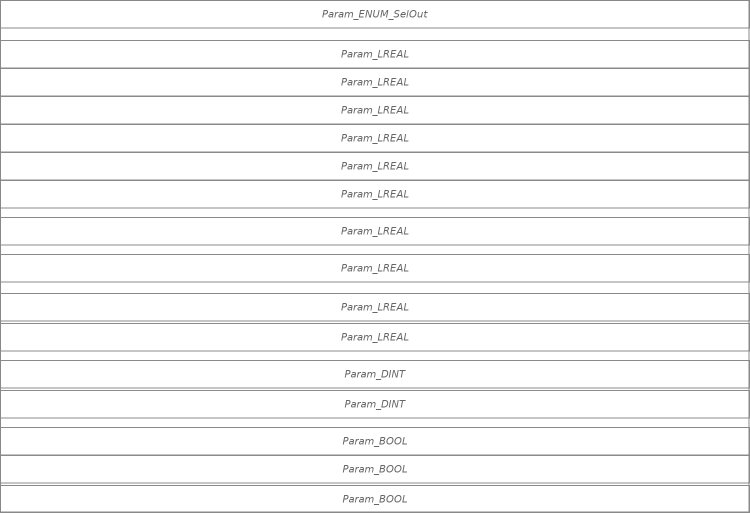
VISUALIZATION Visu_Mparam_Cool  // 750x513
    Frame (0,40 750x28)
        shows Param_LREAL(nIdx := 4)
    Frame (0,68 750x28)
        shows Param_LREAL(nIdx := 6)
    Frame (0,96 750x28)
        shows Param_LREAL(nIdx := 8)
    Frame (0,124 750x28)
        shows Param_LREAL(nIdx := 10)
    Frame (0,360 750x28)
        shows Param_DINT(nIdx := 11)
    Frame (0,0 750x28)
        shows Param_ENUM_SelOut(nIdx := GlobalOne)
    Frame (0,152 750x28)
        shows Param_LREAL(nIdx := 16)
    Frame (0,180 750x28)
        shows Param_LREAL(nIdx := 17)
    Frame (0,217 750x28)
        shows Param_LREAL(nIdx := 21)
    Frame (0,293 750x28)
        shows Param_LREAL(nIdx := 37)
    Frame (0,323 750x28)
        shows Param_LREAL(nIdx := 38)
    Frame (0,427 750x28)
        shows Param_BOOL(nIdx := GlobalOne)
    Frame (0,455 750x28)
        shows Param_BOOL(nIdx := 3)
    Frame (0,485 750x28)
        shows Param_BOOL(nIdx := 18)
    Frame (0,254 750x28)
        shows Param_LREAL(nIdx := 32)
    Frame (0,390 750x28)
        shows Param_DINT(nIdx := 12)
END_VISUALIZATION

(* stored: Version 1.1.0.1
   Visu Visu_Mparam_Cool: Id {4f578426-2293-467e-8b91-0f0781ab1583} *)
